FUNCTION_BLOCK OrchestrationForm2OrchestrationForm (* Helper FB to set the connection to a Orchestration Form type *)
  (* Standard: 61499-2; Description: Copyright (c) 2019 fortiss GmbH This program and the accompanying materials are made available under the terms of the Eclipse Public License 2.0 which is available at https://www.eclipse.org/legal/epl-2.0/ SPDX-License-Identifier: PL-2.0 *)
  (* Version 1.0, 2019-01-28, Jose Cabral, fortiss GmbH *)
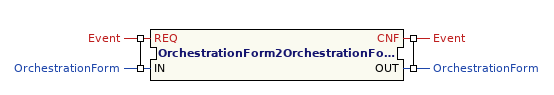
  EVENT_INPUT
    REQ WITH IN; (* Request *)
  END_EVENT
  EVENT_OUTPUT
    CNF WITH OUT; (* Confirm *)
  END_EVENT
  VAR_INPUT
    IN : OrchestrationForm; (* Input *)
  END_VAR
  VAR_OUTPUT
    OUT : OrchestrationForm; (* Output *)
  END_VAR
  (* Service APPLICATION/RESOURCE: Helper FB to set the connection to a Orchestration Form type *)
END_FUNCTION_BLOCK
